# EPICS substitutions: softGlueApp/Db/softGlue_FPGAContent.substitutions
file "softGlue_Input.db"
{
pattern {SIG		ADDR}
{AND-1_IN1		100}
{AND-1_IN2		101}
{AND-2_IN1		102}
{AND-2_IN2		103}
{AND-3_IN1		104}
{AND-3_IN2		105}
{AND-4_IN1		106}
{AND-4_IN2		107}
{OR-1_IN1		108}
{OR-1_IN2		109}
{OR-2_IN1		110}
{OR-2_IN2		111}
{OR-3_IN1		112}
{OR-3_IN2		113}
{OR-4_IN1		114}
{OR-4_IN2		115}
{XOR-1_IN1		116}
{XOR-1_IN2		117}
{XOR-2_IN1		118}
{XOR-2_IN2		119}
{BUFFER-1_IN		120}
{BUFFER-2_IN		121}
{BUFFER-3_IN		122}
{BUFFER-4_IN		123}
{DFF-1_D		124}
{DFF-1_CLOCK		125}
{DFF-1_SET		126}
{DFF-1_CLEAR		127}
{DFF-2_D		128}
{DFF-2_CLOCK		129}
{DFF-2_SET		130}
{DFF-2_CLEAR		131}
{DFF-3_D		132}
{DFF-3_CLOCK		133}
{DFF-3_SET		134}
{DFF-3_CLEAR		135}
{DFF-4_D		136}
{DFF-4_CLOCK		137}
{DFF-4_SET		138}
{DFF-4_CLEAR		139}
{DnCntr-1_ENABLE	140}
{DnCntr-1_CLOCK		141}
{DnCntr-1_LOAD		142}
{DnCntr-2_ENABLE	143}
{DnCntr-2_CLOCK		144}
{DnCntr-2_LOAD		145}
{DnCntr-3_ENABLE	146}
{DnCntr-3_CLOCK		147}
{DnCntr-3_LOAD		148}
{DnCntr-4_ENABLE	149}
{DnCntr-4_CLOCK		150}
{DnCntr-4_LOAD		151}
{UpCntr-1_ENABLE	152}
{UpCntr-1_CLOCK		153}
{UpCntr-1_CLEAR		154}
{UpCntr-2_ENABLE	155}
{UpCntr-2_CLOCK		156}
{UpCntr-2_CLEAR		157}
{UpCntr-3_ENABLE	158}
{UpCntr-3_CLOCK		159}
{UpCntr-3_CLEAR		160}
{UpCntr-4_ENABLE	161}
{UpCntr-4_CLOCK		162}
{UpCntr-4_CLEAR		163}
{DEMUX2-1_IN		164}
{DEMUX2-1_SEL		165}
{DEMUX2-2_IN		166}
{DEMUX2-2_SEL		167}
{MUX2-1_IN0		168}
{MUX2-1_IN1		169}
{MUX2-1_SEL		170}
{MUX2-2_IN0		171}
{MUX2-2_IN1		172}
{MUX2-2_SEL		173}

{DivByN-1_ENABLE	174}
{DivByN-1_CLOCK		175}
{DivByN-1_RESET		176}

{DivByN-2_ENABLE	177}
{DivByN-2_CLOCK		178}
{DivByN-2_RESET		179}

{DivByN-3_ENABLE	180}
{DivByN-3_CLOCK		181}
{DivByN-3_RESET		182}

{DivByN-4_ENABLE	183}
{DivByN-4_CLOCK		184}
{DivByN-4_RESET		185}

{UpDnCntr-1_ENABLE	186}
{UpDnCntr-1_CLOCK	187}
{UpDnCntr-1_LOAD	188}
{UpDnCntr-1_CLEAR	189}
{UpDnCntr-1_UPDOWN	190}

{UpDnCntr-2_ENABLE	191}
{UpDnCntr-2_CLOCK	192}
{UpDnCntr-2_LOAD	193}
{UpDnCntr-2_CLEAR	194}
{UpDnCntr-2_UPDOWN	195}

{UpDnCntr-3_ENABLE	196}
{UpDnCntr-3_CLOCK	197}
{UpDnCntr-3_LOAD	198}
{UpDnCntr-3_CLEAR	199}
{UpDnCntr-3_UPDOWN	200}

{UpDnCntr-4_ENABLE	201}
{UpDnCntr-4_CLOCK	202}
{UpDnCntr-4_LOAD	203}
{UpDnCntr-4_CLEAR	204}
{UpDnCntr-4_UPDOWN	205}

#{UpDnCntr-5_ENABLE	206}
#{UpDnCntr-5_CLOCK	207}
#{UpDnCntr-5_LOAD	208}
#{UpDnCntr-5_CLEAR	209}
#{UpDnCntr-5_UPDOWN	210}

{HistScal-1_EN		206}
{HistScal-1_CLK		207}
{HistScal-1_SYNC	208}
{HistScal-1_DET		209}
{HistScal-1_CLEAR	210}

{QuadDec-1_A		211}
{QuadDec-1_B		212}
{QuadDec-1_CLOCK	213}
{QuadDec-2_A		214}
{QuadDec-2_B		215}
{QuadDec-2_CLOCK	216}
#{MagCmp-1_SAMPLE	217}

{GateDly-1_IN		218}
{GateDly-1_CLK		219}
{GateDly-2_IN		220}
{GateDly-2_CLK		221}
{GateDly-3_IN		222}
{GateDly-3_CLK		223}
{GateDly-4_IN		224}
{GateDly-4_CLK		225}

{shiftM_CLK		226}
{SISO_IN		227}
{SIAO_IN		228}

{FI1	   52}
{FI2	   53}
{FI3	   54}
{FI4	   55}
{FI5	   56}
{FI6	   57}
{FI7	   58}
{FI8	   59}
}

file "softGlue_Output.db"
{
pattern {SIG   	ADDR}

{AND-1_OUT	0}
{AND-2_OUT	1}
{AND-3_OUT	2}
{AND-4_OUT	3}
{OR-1_OUT	4}
{OR-2_OUT	5}
{OR-3_OUT	6}
{OR-4_OUT	7}
{XOR-1_OUT	8}
{XOR-2_OUT	9}
{BUFFER-1_OUT	10}
{BUFFER-2_OUT	11}
{BUFFER-3_OUT	12}
{BUFFER-4_OUT	13}
{DFF-1_OUT	14}
{DFF-2_OUT	15}
{DFF-3_OUT	16}
{DFF-4_OUT	17}
{DnCntr-1_OUT	18}
{DnCntr-2_OUT	19}
{DnCntr-3_OUT	20}
{DnCntr-4_OUT	21}
{DEMUX2-1_OUT0	22}
{DEMUX2-1_OUT1	23}
{DEMUX2-2_OUT0	24}
{DEMUX2-2_OUT1	25}
{MUX2-1_OUT	26}
{MUX2-2_OUT	27}
{DivByN-1_OUT	28}
{DivByN-2_OUT	29}
{DivByN-3_OUT	30}
{DivByN-4_OUT	31}
{UpDnCntr-1_OUT	32}
{UpDnCntr-2_OUT	33}
{UpDnCntr-3_OUT	34}
{UpDnCntr-4_OUT	35}
# Note UpDnCntr-5 is different: OUT->Q8; new output C8
#{UpDnCntr-5_Q8	36}
#{UpDnCntr-5_C8	37}
{QuadDec-1_STEP	38}
{QuadDec-1_DIR	39}
{QuadDec-2_STEP	40}
{QuadDec-2_DIR	41}
#{MagCmp-1_AGTB 42}
#{MagCmp-1_ANEB 43}
#{MagCmp-1_BDIR 44}
#{MagCmp-1_BCK  45}
{40MHZ_CLOCK	46}
{10MHZ_CLOCK	47}
{GateDly-1_OUT	48}
{GateDly-2_OUT	49}
{GateDly-3_OUT	50}
{GateDly-4_OUT	51}

{AISO_OUT		36}
{SISO_OUT		37}

{FO1   231}
{FO2   232}
{FO3   233}
{FO4   234}
{FO5   235}
{FO6   236}
{FO7   237}
{FO8   238}

}

#file "softGlue_FieldInput.db"
#{
#pattern {SIG   PORT	ADDR       IOPIN}
## These are inputs from the user's viewpoint, but they behave like softGlue
## outputs.
#{FI1	   52}
#{FI2	   53}
#{FI3	   54}
#{FI4	   55}
#{FI5	   56}
#{FI6	   57}
#{FI7	   58}
#{FI8	   59}
#{FI9	    9}
#{FI10		10}
#{FI11		11}
#{FI12		12}
#{FI13		13}
#{FI14		14}
#{FI15		15}
#{FI16		16}
#{FI17		17}
#{FI18		18}
#{FI19		19}
#{FI20		20}
#{FI21		21}
#{FI22		22}
#{FI23		23}
#{FI24		24}
#{FI25		25}
#{FI26		26}
#{FI27		27}
#{FI28		28}
#{FI29		29}
#{FI30		30}
#{FI31		31}
#{FI32		32}
#{FI33		33}
#{FI34		34}
#{FI35		35}
#{FI36		36}
#{FI37		37}
#{FI38		38}
#{FI39		39}
#{FI40		40}
#{FI41		41}
#{FI42		42}
#{FI43		43}
#{FI44		44}
#{FI45		45}
#{FI46		46}
#{FI47		47}
#{FI48		48}
#}

#file "softGlue_FieldOutput.db"
#{
#pattern {SIG   ADDR       IOPIN}
## These are outputs from the user's viewpoint, but they behave like softGlue
## inputs.
#{FO1   231}
#{FO2   232}
#{FO3   233}
#{FO4   234}
#{FO5   235}
#{FO6   236}
#{FO7   237}
#{FO8   238}
#{FO9	9}
#{FO10	10}
#{FO11	11}
#{FO12	12}
#{FO13	13}
#{FO14	14}
#{FO15	15}
#{FO16	16}
#{FO17	17}
#{FO18	18}
#{FO19	19}
#{FO20	20}
#{FO21	21}
#{FO22	22}
#{FO23	23}
#{FO24	24}
#{FO25	25}
#{FO26	26}
#{FO27	27}
#{FO28	28}
#{FO29	29}
#{FO30	30}
#{FO31	31}
#{FO32	32}
#{FO33	33}
#{FO34	34}
#{FO35	35}
#{FO36	36}
#{FO37	37}
#{FO38	38}
#{FO39	39}
#{FO40	40}
#{FO41	41}
#{FO42	42}
#{FO43	43}
#{FO44	44}
#{FO45	45}
#{FO46	46}
#{FO47	47}
#{FO48	48}
#}

file "softGlue_description.db"
{
pattern {SIG N}
{circuit 300}
{10MHZ_CLOCK 80}
{40MHZ_CLOCK 80}
{800MHZ_CLOCK 80}
{AND-1 80}
{AND-2 80}
{AND-3 80}
{AND-4 80}
{OR-1 80}
{OR-2 80}
{OR-3 80}
{OR-4 80}
{XOR-1 80}
{XOR-2 80}
{BUFFER-1 80}
{BUFFER-2 80}
{BUFFER-3 80}
{BUFFER-4 80}
{DEMUX2-1 80}
{DEMUX2-2 80}
{DFF-1 80}
{DFF-2 80}
{DFF-3 80}
{DFF-4 80}
{DivByN-1 80}
{DivByN-2 80}
{DivByN-3 80}
{DivByN-4 80}
{DnCntr-1 80}
{DnCntr-2 80}
{DnCntr-3 80}
{DnCntr-4 80}
{MUX2-1 80}
{MUX2-2 80}
{UpCntr-1 80}
{UpCntr-2 80}
{UpCntr-3 80}
{UpCntr-4 80}
{UpDnCntr-1 80}
{UpDnCntr-2 80}
{UpDnCntr-3 80}
{UpDnCntr-4 80}
{UpDnCntr-5 80}
{QuadDec-1 80}
{QuadDec-2 80}
{MagCmp-1 80}
#{HistScal-1 80}
}

# pinout:
# sig	zynqP	zynqN	mzedP	mzedN	bkoutP	bkoutN
#			JX1	JX1	CON1	CON1
#---------------------------------------------------------
# FI1	T11	T10	11	13	5	7
# FI2	T12	U12	12	14	6	8
# FI3	U13	V13	17	19	9	11
# FI4	V12	W13	18	20	10	12
# FI5	T14	T15	23	25	13	15
# FI6	P14	R14	24	26	14	16
# FI7	Y16	Y17	29	31	19	21
# FI8	W14	Y14	30	32	20	22
# FI9	T16	U17	35	37	23	25
# FI10	V15	W15	36	38	24	26
# FI11	U14	U15	41	43	27	29
# FI12	U18	U19	42	44	28	30
#
# FO1	N18	P19	47	49	31	33
# FO2	N20	P20	48	50	32	34
# FO3	T20	U20	53	55	35	37
# FO4	V20	W20	54	56	36	38
# FO5	Y18	Y19	61	63	41	43
# FO6	V16	W16	62	64	42	44
# FO7	R16	R17	67	69	45	47
# FO8	T17	R18	68	70	46	48
# FO9	V17	V18	73	75	49	51
# FO10	W18	W19	74	76	50	52
# FO11	N17	P18	81	83	55	57
# FO12	P15	P16	82	84	56	58
